// TIA Portal V16 export
// export: Created 2024-12-03T15:41:40.196613Z, ExportSetting WithDefaults, DisplayName Totally Integrated Automation Portal, DisplayVersion V16 Update 6, DisplayName TIA Portal Version Control Interface, DisplayVersion V16 Update 2, DisplayName TIA Portal Openness, DisplayVersion V16 Update 6, DisplayName TIA Portal Teamcenter Gateway, DisplayVersion V16, DisplayName SINAMICS Startdrive Advanced, DisplayVersion V16 Update 5, DisplayName SINAMICS Startdrive G130, G150, S120, S150, SINAMICS MV, S210, DisplayVersion V16 Update 5, DisplayName SINAMICS Startdrive G110M, G120, G120C, G120D, G120P, G115D, DisplayVersion V16 Update 5, DisplayName STEP 7 Professional, DisplayVersion V16 Update 6, DisplayName STEP 7 Safety, DisplayVersion V16, DisplayName WinCC Advanced / Unified PC, DisplayVersion V16 Update 6
FUNCTION_BLOCK "Z_100_INTERFACE_FB"   // FB74, SCL
{ S7_Optimized_Access := 'TRUE' }
VERSION : 0.1
// stored: AutoNumber true, IsIECCheckEnabled false, IsRetainMemResEnabled false, MemoryReserve 100, SetENOAutomatically false, UDAEnableTagReadback false
BEGIN
   REGION LOOP

       REGION CONV_101

           "Motor_Conveyor_Interface"(
                                      I_RunningFeedback := "DRV_DB".DRV_101_DRV_1.Status.Running,
                                      I_MotorAlarm := FALSE,
                                      IO_SensorStart := "Inputs_DB".FTC_115_L2,
                                      IO_SensorEnd := "Inputs_DB".FTC_102_L2,
                                      IO_Conveyor := "CONV_DB".CONV_101);

       END_REGION

       REGION CONV_102L

           "Motor_Conveyor_Interface"(
                                      I_RunningFeedback := "MOT_CLX_DB".MOT_102L.Status.Running,
                                      I_MotorAlarm := FALSE,
                                      IO_SensorStart := "Inputs_DB".FTC_102_L2,
                                      IO_SensorEnd := "Inputs_DB".FTC_102_L4,
                                      IO_Conveyor := "CONV_DB".CONV_102L);

       END_REGION

       REGION CONV_102R

           "Motor_Conveyor_Interface"(
                                      I_RunningFeedback := "MOT_CLX_DB".MOT_102R.Status.Running,
                                      I_MotorAlarm := FALSE,
                                      IO_SensorStart := "Inputs_DB".FTC_102_L4,
                                      IO_SensorEnd := "Inputs_DB".FTC_102_R4,
                                      IO_Conveyor := "CONV_DB".CONV_102R);

       END_REGION

       REGION CONV_103L

           "Motor_Conveyor_Interface"(
                                      I_RunningFeedback := "MOT_CLX_DB".MOT_103L.Status.Running,
                                      I_MotorAlarm := FALSE,
                                      IO_SensorStart := "Inputs_DB".FTC_102_R4,
                                      IO_SensorEnd := "Inputs_DB".FTC_103_L4,
                                      IO_Conveyor := "CONV_DB".CONV_103L);

       END_REGION

       REGION CONV_103R

           "Motor_Conveyor_Interface"(
                                      I_RunningFeedback := "MOT_CLX_DB".MOT_103R.Status.Running,
                                      I_MotorAlarm := FALSE,
                                      IO_SensorStart := "Inputs_DB".FTC_103_L4,
                                      IO_SensorEnd := "Inputs_DB".FTC_103_R4,
                                      IO_Conveyor := "CONV_DB".CONV_103R);

       END_REGION

       REGION CONV_104R

           "Motor_Conveyor_Interface"(
                                      I_RunningFeedback := "MOT_CLX_DB".MOT_104R.Status.Running,
                                      I_MotorAlarm := FALSE,
                                      IO_SensorStart := "Inputs_DB".FTC_103_R4,
                                      IO_SensorEnd := "Inputs_DB".FTC_104_R4,
                                      IO_Conveyor := "CONV_DB".CONV_104R);

       END_REGION

       REGION CONV_104L

           "Motor_Conveyor_Interface"(
                                      I_RunningFeedback := "MOT_CLX_DB".MOT_104L.Status.Running,
                                      I_MotorAlarm := FALSE,
                                      IO_SensorStart := "Inputs_DB".FTC_104_R4,
                                      IO_SensorEnd := "Inputs_DB".FTC_104_L4,
                                      IO_Conveyor := "CONV_DB".CONV_104L);

       END_REGION

       REGION CONV_105R

           "Motor_Conveyor_Interface"(
                                      I_RunningFeedback := "MOT_CLX_DB".MOT_105R.Status.Running,
                                      I_MotorAlarm := FALSE,
                                      IO_SensorStart := "Inputs_DB".FTC_104_L4,
                                      IO_SensorEnd := "Inputs_DB".FTC_105_R4,
                                      IO_Conveyor := "CONV_DB".CONV_105R);

       END_REGION

       REGION CONV_105L

           "Motor_Conveyor_Interface"(
                                      I_RunningFeedback := "MOT_CLX_DB".MOT_105L.Status.Running,
                                      I_MotorAlarm := FALSE,
                                      IO_SensorStart := "Inputs_DB".FTC_105_R4,
                                      IO_SensorEnd := "Inputs_DB".FTC_105_L4,
                                      IO_Conveyor := "CONV_DB".CONV_105L);

       END_REGION

       REGION CONV_106R

           "Motor_Conveyor_Interface"(
                                      I_RunningFeedback := "MOT_CLX_DB".MOT_106R.Status.Running,
                                      I_MotorAlarm := FALSE,
                                      IO_SensorStart := "Inputs_DB".FTC_105_L4,
                                      IO_SensorEnd := "Inputs_DB".FTC_106_R4,
                                      IO_Conveyor := "CONV_DB".CONV_106R);

       END_REGION

       REGION CONV_107R

           "Motor_Conveyor_Interface"(
                                      I_RunningFeedback := "MOT_CLX_DB".MOT_107R.Status.Running AND "MOT_CLX_DB".MOT_106L.Status.Running,
                                      I_MotorAlarm := FALSE,
                                      IO_SensorStart := "Inputs_DB".FTC_106_R4,
                                      IO_SensorEnd := "Inputs_DB".FTC_106_L4,
                                      IO_Conveyor := "CONV_DB".CONV_107R);

       END_REGION

       REGION CONV_108R

           "Motor_Conveyor_Interface"(
                                      I_RunningFeedback := "MOT_CLX_DB".MOT_108R.Status.Running,
                                      I_MotorAlarm := FALSE,
                                      IO_SensorStart := "Inputs_DB".FTC_106_L4,
                                      IO_SensorEnd := "Inputs_DB".FTC_108_R4,
                                      IO_Conveyor := "CONV_DB".CONV_108R);

       END_REGION

       REGION CONV_108L

           "Motor_Conveyor_Interface"(
                                      I_RunningFeedback := "MOT_CLX_DB".MOT_108L.Status.Running,
                                      I_MotorAlarm := FALSE,
                                      IO_SensorStart := "Inputs_DB".FTC_108_R4,
                                      IO_SensorEnd := "Inputs_DB".FTC_108_L4,
                                      IO_Conveyor := "CONV_DB".CONV_108L);

       END_REGION

       REGION CONV_109R

           "Motor_Conveyor_Interface"(
                                      I_RunningFeedback := "MOT_CLX_DB".MOT_109R.Status.Running,
                                      I_MotorAlarm := FALSE,
                                      IO_SensorStart := "Inputs_DB".FTC_108_L4,
                                      IO_SensorEnd := "Inputs_DB".FTC_109_R4,
                                      IO_Conveyor := "CONV_DB".CONV_109R);

       END_REGION

       REGION CONV_109L

           "Motor_Conveyor_Interface"(
                                      I_RunningFeedback := "MOT_CLX_DB".MOT_109L.Status.Running,
                                      I_MotorAlarm := FALSE,
                                      IO_SensorStart := "Inputs_DB".FTC_109_R4,
                                      IO_SensorEnd := "Inputs_DB".FTC_109_L4,
                                      IO_Conveyor := "CONV_DB".CONV_109L);

       END_REGION

       REGION CONV_110R

           "Motor_Conveyor_Interface"(
                                      I_RunningFeedback := "MOT_CLX_DB".MOT_110R.Status.Running,
                                      I_MotorAlarm := FALSE,
                                      IO_SensorStart := "Inputs_DB".FTC_109_L4,
                                      IO_SensorEnd := "Inputs_DB".FTC_110_R4,
                                      IO_Conveyor := "CONV_DB".CONV_110R);

       END_REGION

       REGION CONV_110L

           "Motor_Conveyor_Interface"(
                                      I_RunningFeedback := "MOT_CLX_DB".MOT_110L.Status.Running,
                                      I_MotorAlarm := FALSE,
                                      IO_SensorStart := "Inputs_DB".FTC_110_R4,
                                      IO_SensorEnd := "Inputs_DB".FTC_110_L4,
                                      IO_Conveyor := "CONV_DB".CONV_110L);

       END_REGION

       REGION TRANSFER CONV 111R

           REGION CONV_111R 

               "Motor_Conveyor_Interface"(
                                          I_RunningFeedback := "MOT_CLX_DB".MOT_111R.Status.Running,
                                          I_MotorAlarm := FALSE,
                                          IO_SensorStart := "Inputs_DB".FTC_110_L4,
                                          IO_SensorEnd := "Inputs_DB".FTC_111_R4,
                                          IO_Conveyor := "CONV_DB".CONV_111R);

           END_REGION

           REGION CONV_201R_BELTS

               "Motor_Conveyor_Interface"(
                                          I_RunningFeedback := "MOT_CLX_DB".MOT_201R_Belts.Status.Running,
                                          I_MotorAlarm := FALSE,
                                          IO_SensorStart := "Inputs_DB".FTC_111_R4,
                                          IO_SensorEnd := "Inputs_DB".FTC_111_R4,
                                          IO_Conveyor := "CONV_DB".CONV_201R_BELTS);

           END_REGION

       END_REGION

       REGION CONV_111L

           "Motor_Conveyor_Interface"(
                                      I_RunningFeedback := "MOT_CLX_DB".MOT_111L.Status.Running,
                                      I_MotorAlarm := FALSE,
                                      IO_SensorStart := "Inputs_DB".FTC_111_R4,
                                      IO_SensorEnd := "Inputs_DB".FTC_111_L4,
                                      IO_Conveyor := "CONV_DB".CONV_111L);

       END_REGION

       REGION CONV_112R

           "Motor_Conveyor_Interface"(
                                      I_RunningFeedback := "MOT_CLX_DB".MOT_112R.Status.Running,
                                      I_MotorAlarm := FALSE,
                                      IO_SensorStart := "Inputs_DB".FTC_111_L4,
                                      IO_SensorEnd := "Inputs_DB".FTC_112_R4,
                                      IO_Conveyor := "CONV_DB".CONV_112R);

       END_REGION

       REGION CONV_113L

           "Motor_Conveyor_Interface"(
                                      I_RunningFeedback := "MOT_CLX_DB".MOT_113L.Status.Running AND "MOT_CLX_DB".MOT_112L.Status.Running,
                                      I_MotorAlarm := FALSE,
                                      IO_SensorStart := "Inputs_DB".FTC_112_R4,
                                      IO_SensorEnd := "Inputs_DB".FTC_113_L4,
                                      IO_Conveyor := "CONV_DB".CONV_113L);

       END_REGION

       REGION CONV_114R

           "Motor_Conveyor_Interface"(
                                      I_RunningFeedback := "MOT_CLX_DB".MOT_114R.Status.Running,
                                      I_MotorAlarm := FALSE,
                                      IO_SensorStart := "Inputs_DB".FTC_113_L4,
                                      IO_SensorEnd := "Inputs_DB".FTC_114_R4,
                                      IO_Conveyor := "CONV_DB".CONV_114R);

       END_REGION

       REGION CONV_114L

           "Motor_Conveyor_Interface"(
                                      I_RunningFeedback := "MOT_CLX_DB".MOT_114L.Status.Running,
                                      I_MotorAlarm := FALSE,
                                      IO_SensorStart := "Inputs_DB".FTC_114_R4,
                                      IO_SensorEnd := "Inputs_DB".FTC_114_L4,
                                      IO_Conveyor := "CONV_DB".CONV_114L);

       END_REGION

       REGION CONV_115R

           "Motor_Conveyor_Interface"(
                                      I_RunningFeedback := "MOT_CLX_DB".MOT_115R.Status.Running,
                                      I_MotorAlarm := FALSE,
                                      IO_SensorStart := "Inputs_DB".FTC_114_L4,
                                      IO_SensorEnd := "Inputs_DB".FTC_115_R4,
                                      IO_Conveyor := "CONV_DB".CONV_115R);

       END_REGION

       REGION CONV_115L

           "Motor_Conveyor_Interface"(
                                      I_RunningFeedback := "MOT_CLX_DB".MOT_115L.Status.Running,
                                      I_MotorAlarm := FALSE,
                                      IO_SensorStart := "Inputs_DB".FTC_115_R4,
                                      IO_SensorEnd := "Inputs_DB".FTC_115_L4,
                                      IO_Conveyor := "CONV_DB".CONV_115L);

       END_REGION


   END_REGION

   REGION SIDE LANE

       REGION CONV_301R

           "Motor_Conveyor_Interface"(
                                      I_RunningFeedback := "MOT_CLX_DB".MOT_301R.Status.Running AND "MOT_CLX_DB".MOT_301L.Status.Running,
                                      I_MotorAlarm := FALSE,
                                      IO_SensorStart := "Inputs_DB".FTC_106_L4,
                                      IO_SensorEnd := "Inputs_DB".FTC_301_R4,
                                      IO_Conveyor := "CONV_DB".CONV_301R);

       END_REGION

       REGION CONV_302L

           "Motor_Conveyor_Interface"(
                                      I_RunningFeedback := "MOT_CLX_DB".MOT_302L.Status.Running,
                                      I_MotorAlarm := FALSE,
                                      IO_SensorStart := "Inputs_DB".FTC_301_R4,
                                      IO_SensorEnd := "Inputs_DB".FTC_302_L4,
                                      IO_Conveyor := "CONV_DB".CONV_302L);

       END_REGION

       REGION CONV_302R

           "Motor_Conveyor_Interface"(
                                      I_RunningFeedback := "MOT_CLX_DB".MOT_302R.Status.Running,
                                      I_MotorAlarm := FALSE,
                                      IO_SensorStart := "Inputs_DB".FTC_302_L4,
                                      IO_SensorEnd := "Inputs_DB".FTC_302_R4,
                                      IO_Conveyor := "CONV_DB".CONV_302R);

       END_REGION

       REGION CONV_303L

           "Motor_Conveyor_Interface"(
                                      I_RunningFeedback := "MOT_CLX_DB".MOT_303L.Status.Running,
                                      I_MotorAlarm := FALSE,
                                      IO_SensorStart := "Inputs_DB".FTC_302_R4,
                                      IO_SensorEnd := "Inputs_DB".FTC_303_L4,
                                      IO_Conveyor := "CONV_DB".CONV_303L);

       END_REGION

       REGION CONV_303R

           "Motor_Conveyor_Interface"(
                                      I_RunningFeedback := "MOT_CLX_DB".MOT_303R.Status.Running,
                                      I_MotorAlarm := FALSE,
                                      IO_SensorStart := "Inputs_DB".FTC_303_L4,
                                      IO_SensorEnd := "Inputs_DB".FTC_303_R4,
                                      IO_Conveyor := "CONV_DB".CONV_303R);

       END_REGION

       REGION TRANSFER

           REGION CONV_304L

               "Motor_Conveyor_Interface"(
                                          I_RunningFeedback := "MOT_CLX_DB".MOT_304L.Status.Running,
                                          I_MotorAlarm := FALSE,
                                          IO_SensorStart := "Inputs_DB".FTC_303_R4,
                                          IO_SensorEnd := "Inputs_DB".FTC_304_L4,
                                          IO_Conveyor := "CONV_DB".CONV_304L);

           END_REGION

           REGION CONV_304L

               "Motor_Conveyor_Interface"(
                                          I_RunningFeedback := "MOT_CLX_DB".MOT_304L.Status.Running AND
                                          "MOT_CLX_DB".MOT_202L.Status.Running AND
                                          "MOT_CLX_DB".MOT_202R.Status.Running,
                                          I_MotorAlarm := FALSE,
                                          IO_SensorStart :="Inputs_DB".FTC_304_L4,
                                          IO_SensorEnd := "Inputs_DB".FTC_304_L4,
                                          IO_Conveyor := "CONV_DB".CONV_304L);

           END_REGION

       END_REGION

       REGION CONV_304R

           "Motor_Conveyor_Interface"(
                                      I_RunningFeedback := "MOT_CLX_DB".MOT_304R.Status.Running,
                                      I_MotorAlarm := FALSE,
                                      IO_SensorStart := "Inputs_DB".FTC_304_L4,
                                      IO_SensorEnd := "Inputs_DB".FTC_304_R4,
                                      IO_Conveyor := "CONV_DB".CONV_304R);

       END_REGION

       REGION CONV_305R

           "Motor_Conveyor_Interface"(
                                      I_RunningFeedback := "MOT_CLX_DB".MOT_305R.Status.Running AND "MOT_CLX_DB".MOT_305L.Status.Running,
                                      I_MotorAlarm := FALSE,
                                      IO_SensorStart := "Inputs_DB".FTC_304_R4, //"Inputs_DB".FTC_305_L4,
                                      IO_SensorEnd := "Inputs_DB".FTC_305_R4,
                                      IO_Conveyor := "CONV_DB".CONV_305R);

       END_REGION

   END_REGION
END_FUNCTION_BLOCK
